(*
Implements the procedure for safely transitioning between device states by asserting the correct beam parameters for 
the state *)
FUNCTION_BLOCK BeamClassTransitionManager
VAR_INPUT
	i_stTransitionAssertion : ST_BeamParams; //Assertion required during transition (always safer than anything inbetween)
	i_stFinalAssertion	:	ST_BeamParams; //Assertion required after transition
	i_xMoving	:	BOOL; //Provide rising edge when device begins moving
	i_xDoneMoving	:	BOOL; //Provide rising edge when device is done with a move
	i_stFullBeam	:	ST_BeamParams := PMPS_GVL_BeamParams.cstFullBeam; //Beam parameters applied to transition assertion once transition is complete
END_VAR
VAR_OUTPUT
	q_stTransitionAssertion	:	ST_BeamParams; //Transition assertion
	q_stFinalAssertion	:	ST_BeamParams; //Final assertion
	q_MoveAuthorized	:	BOOL; //Rising edge indicating the device is safe to move, use as input to move execute (which requires a rising edge)
END_VAR
VAR
END_VAR

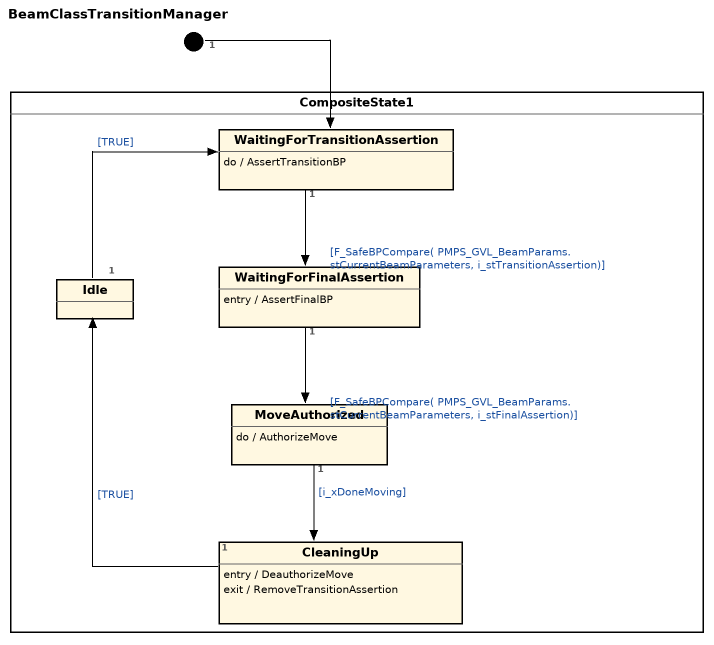
STATECHART ExampleSC  // abortable
    START StartState1
    COMPOSITE STATE CompositeState1
        STATE WaitingForTransitionAssertion
            do / AssertTransitionBP
        STATE Idle
        STATE WaitingForFinalAssertion
            entry / AssertFinalBP
        STATE MoveAuthorized
            do / AuthorizeMove
        STATE CleaningUp
            entry / DeauthorizeMove
            exit / RemoveTransitionAssertion
        WaitingForTransitionAssertion -> WaitingForFinalAssertion [F_SafeBPCompare( PMPS_GVL_BeamParams.stCurrentBeamParameters, i_stTransitionAssertion)] // priority 1
        Idle -> WaitingForTransitionAssertion [TRUE] // priority 1
        WaitingForFinalAssertion -> MoveAuthorized [F_SafeBPCompare( PMPS_GVL_BeamParams.stCurrentBeamParameters, i_stFinalAssertion)] // priority 1
        MoveAuthorized -> CleaningUp [i_xDoneMoving] // priority 1, rising edge
        CleaningUp -> Idle [TRUE] // priority 1
    END_STATE
    StartState1 -> WaitingForTransitionAssertion  // priority 1, on completion
END_STATECHART

ACTION AssertFinalBP:
q_stFinalAssertion := i_stFinalAssertion;
END_ACTION

ACTION AssertTransitionBP:
q_stTransitionAssertion := i_stTransitionAssertion;
END_ACTION

ACTION AuthorizeMove:
q_MoveAuthorized := TRUE;
END_ACTION

ACTION DeauthorizeMove:
q_MoveAuthorize := FALSE;
END_ACTION

ACTION RemoveTransitionAssertion:
q_stTransitionAssertion = cstFullBeam;
END_ACTION

END_FUNCTION_BLOCK

(* stored: Version 1.1.0.1, ProductVersion 3.1.4022.12
   POU BeamClassTransitionManager: Id {0bd0e55a-9cb3-42b8-83b7-fffcea3ac6a4}, SpecialFunc None
   Action AssertFinalBP: Id {01eff59d-4502-4abf-a177-909c4feb4c0d}
   Action AssertTransitionBP: Id {ee0b045b-0e87-4101-b654-13a82bd0baba}
   Action AuthorizeMove: Id {891b1b7e-92c0-4a6e-97f0-de00417e3c3d}
   Action DeauthorizeMove: Id {c50e542b-a4ee-42b6-86ca-efb3051c4d56}
   Action RemoveTransitionAssertion: Id {81e3a5bb-9ce0-4ae8-b3c5-d28719247253} *)
